{attribute 'qualified_only'}
VAR_GLOBAL CONSTANT
    cErrorHistMin : INT := 0; ///Error history array bound minimum
    cErrorHistMax : INT := 10; ///Error history array bound maximum
END_VAR

(* stored: Version 1.1.0.1, ProductVersion 3.1.4019.2
   GVL GVL_ObjectSetup: Id {518ef158-1f4f-4831-a267-9e7c804cab79} *)
